// TIA Portal V15.1 export
// export: Created 2026-01-15T16:29:46.2078086Z, ExportSetting WithDefaults, WithReadOnly, DisplayName Totally Integrated Automation Portal, DisplayVersion V15.1 Update 8, DisplayName TIA Portal Openness, DisplayVersion V15.1 Update 8, DisplayName STEP 7 Professional, DisplayVersion V15.1 Update 8, DisplayName WinCC Advanced, DisplayVersion V15.1 Update 8
DATA_BLOCK "C#7_RD_RUN"   // DB7
{ S7_Optimized_Access := 'FALSE' }
VERSION : 0.1
// stored: AutoNumber true, CodeModifiedDate 2026-01-10T14:48:41.7878153Z, CompileDate 2026-01-15T16:25:51.9514339Z, CreationDate 2026-01-15T16:23:32.6582836Z, DBAccessibleFromOPCUA true, InterfaceModifiedDate 2026-01-10T14:48:41.7878153Z, IsConsistent true, IsKnowHowProtected false, IsOnlyStoredInLoadMemory false, IsPLCDB false, IsWriteProtectedInAS false, ModifiedDate 2026-01-12T11:40:02.1103777Z, ParameterModified 2026-01-10T14:48:41.7878153Z, StructureModified 2026-01-10T14:48:41.7878153Z
   VAR RETAIN
      PV_AG1 : Real;   // Thực cân cốt liệu 1
      "%_WAG1" : Real;   // Phần trăm khối lượng cốt liệu 1
      WE_AG1 : Real;   // Khối lượng cân cốt liệu 1
      SMC_AG1 : Real;   // Số mẻ cân phễu cân cốt liệu 1
      SMX_AG1 : Real;   // Số mẻ xả phễu cân cốt liệu 1
      PV_AG2 : Real;   // Thực cân cốt liệu 2
      SMC_AG2 : Real;   // Số mẻ cân phễu cân cốt liệu 2
      SMX_AG2 : Real;   // Số mẻ xả phễu cân cốt liệu 2
      PV_AG3 : Real;   // Thực cân cốt liệu 3
      SMC_AG3 : Real;   // Số mẻ cân phễu cân cốt liệu 3
      SMX_AG3 : Real;   // Số mẻ xả phễu cân cốt liệu 3
      PV_AG4 : Real;   // Thực cân cốt liệu 4
      SMC_AG4 : Real;   // Số mẻ cân phễu cân cốt liệu 4
      SMX_AG4 : Real;   // Số mẻ xả phễu cân cốt liệu 4
      PV_AG5 : Real;   // Thực cân cốt liệu 5
      SMC_AG5 : Real;   // Số mẻ cân phễu cân cốt liệu 5
      SMX_AG5 : Real;   // Số mẻ xả phễu cân cốt liệu 5
      PV_FD1 : Real;   // Thực cân silo FD 1
      "%_WFD1" : Real;   // Phần trăm khối lượng phễu cân FD 1
      WE_FD1 : Real;   // Khối lượng phễu cân FD 1
      SMC_FD1 : Real;   // Số mẻ cân phễu cân FD 1
      SMX_FD1 : Real;   // Số mẻ xả phễu cân FD 1
      PV_AP1 : Real;   // Thực cân Nhựa 1
      "%_WAP1" : Real;   // Phần trăm khối lượng phễu cân Nhựa 1
      WE_AP1 : Real;   // Khối lượng phễu cân Nhựa 1
      SMC_AP1 : Real;   // Số mẻ cân phễu cân Nhựa 1
      SMX_AP1 : Real;   // Số mẻ xả phễu cân Nhựa 1
      PV_SB1 : Real;   // Thực cân SBS 1
      "%_WSB1" : Real;   // Phần trăm khối lượng phễu cân SBS 1
      WE_SB1 : Real;   // Khối lượng phễu cân SBS 1
      SMC_SB1 : Real;   // Số mẻ cân phễu cân SBS 1
      SMX_SB1 : Real;   // Số mẻ xả phễu cân SBS 1
      SMC_MIXER : Real;   // Số mẻ cân nồi trộn, sẽ tăng lên 1 khi nạp đủ các thành phần liệu
      SMX_MIXER : Real;   // Số mẻ xả nồi trộn
      "TG_THUC TRON" : Real;   // Thoi gian thuc tron
      TG_THUC_XA : Real;   // Thoi gian thuc xa
      SMT : Real;
      "M3/ME" : Real;
      PVM_AG1 : Real;   // Thực cân tay cốt liệu 1
      PVM_AG2 : Real;   // Thực cân tay cốt liệu 2
      PVM_AG3 : Real;   // Thực cân tay cốt liệu 3
      PVM_AG4 : Real;   // Thực cân tay cốt liệu 4
      PVM_AG5 : Real;   // Thực cân tay cốt liệu 5
      PVM_FD1 : Real;   // Thực cân tay FD1
      PVM_AP1 : Real;   // Thực cân tay Nhựa
      PVM_SB1 : Real;   // Thực cân tay SBS1
      TEMP_TUILOC : Real;   // Nhiệt độ túi lọc hiển thị
      TEMP_AGG : Real;   // Nhiệt độ cốt liệu hiển thị
      TEMP_TANSAY : Real;   // Nhiệt độ tan sấy hiển thị
      TEMP_NHUA : Real;   // Nhiệt độ nhựa hiển thị
      WE_AG2 : Real;   // Khối lượng cân cốt liệu 2
      WE_AG3 : Real;   // Khối lượng cân cốt liệu 3
      WE_AG4 : Real;   // Khối lượng cân cốt liệu 4
      WE_AG5 : Real;   // Khối lượng cân cốt liệu 5
      "%_WAG2" : Real;   // Phần trăm khối lượng cốt liệu 2
      "%_WAG3" : Real := 0.0;   // Phần trăm khối lượng cốt liệu 3
      "%_WAG4" : Real := 0.0;   // Phần trăm khối lượng cốt liệu 4
      "%_WAG5" : Real := 0.0;   // Phần trăm khối lượng cốt liệu 5
   END_VAR
BEGIN
END_DATA_BLOCK
